FUNCTION_BLOCK FB_CTRL_PID (* Composite Function Block Type *)
  (* Standard: 61499-2 *)
  (* Version 0.0, 2013-10-19, 4DIAC-IDE, 4DIAC-Consortium *)
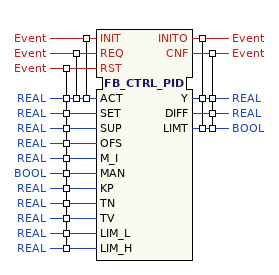
  EVENT_INPUT
    INIT WITH ACT; (* Initialization Request *)
    REQ WITH ACT; (* Normal Execution Request *)
    RST WITH ACT, SET, SUP, OFS, M_I, MAN, KP, TN, TV, LIM_L, LIM_H;
  END_EVENT
  EVENT_OUTPUT
    INITO WITH Y, LIMT; (* Initialization Confirm *)
    CNF WITH Y, DIFF, LIMT; (* Execution Confirmation *)
  END_EVENT
  VAR_INPUT
    ACT : REAL; (* Input event qualifier *)
    SET : REAL; (* default *)
    SUP : REAL; (* noise reduction *)
    OFS : REAL; (* offeset for the output *)
    M_I : REAL; (* input value for manual operation *)
    MAN : BOOL; (* switch to manual mode *)
    KP : REAL; (* controller gain *)
    TN : REAL; (* reset of the controller *)
    TV : REAL; (* derivative of the controller *)
    LIM_L : REAL; (* lower output limit *)
    LIM_H : REAL; (* upper output limit *)
  END_VAR
  VAR_OUTPUT
    Y : REAL; (* output of the controller *)
    DIFF : REAL; (* deviation *)
    LIMT : BOOL; (* TRUE if the output has reached a limit *)
  END_VAR
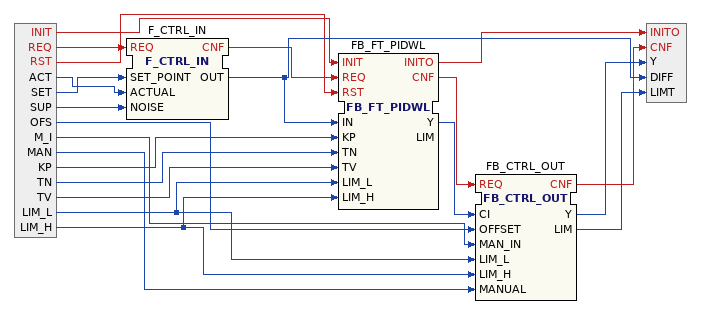
  FBS
    F_CTRL_IN : F_CTRL_IN;
    FB_FT_PIDWL : FB_FT_PIDWL;
    FB_CTRL_OUT : FB_CTRL_OUT;
  END_FBS
  EVENT_CONNECTIONS
    REQ TO F_CTRL_IN.REQ;
    INIT TO FB_FT_PIDWL.INIT;
    RST TO FB_FT_PIDWL.RST;
    F_CTRL_IN.CNF TO FB_FT_PIDWL.REQ;
    FB_FT_PIDWL.INITO TO INITO;
    FB_FT_PIDWL.CNF TO FB_CTRL_OUT.REQ;
    FB_CTRL_OUT.CNF TO CNF;
  END_CONNECTIONS
  DATA_CONNECTIONS
    F_CTRL_IN.OUT TO DIFF;
    SET TO F_CTRL_IN.SET_POINT;
    ACT TO F_CTRL_IN.ACTUAL;
    SUP TO F_CTRL_IN.NOISE;
    F_CTRL_IN.OUT TO FB_FT_PIDWL.IN;
    KP TO FB_FT_PIDWL.KP;
    TN TO FB_FT_PIDWL.TN;
    TV TO FB_FT_PIDWL.TV;
    LIM_L TO FB_FT_PIDWL.LIM_L;
    LIM_H TO FB_FT_PIDWL.LIM_H;
    FB_CTRL_OUT.Y TO Y;
    FB_CTRL_OUT.LIM TO LIMT;
    FB_FT_PIDWL.Y TO FB_CTRL_OUT.CI;
    OFS TO FB_CTRL_OUT.OFFSET;
    M_I TO FB_CTRL_OUT.MAN_IN;
    MAN TO FB_CTRL_OUT.MANUAL;
    LIM_L TO FB_CTRL_OUT.LIM_L;
    LIM_H TO FB_CTRL_OUT.LIM_H;
  END_CONNECTIONS
END_FUNCTION_BLOCK
